FUNCTION_BLOCK FB_HwRefStopButton
VAR_INPUT
END_VAR
VAR_OUTPUT
END_VAR
VAR
	bInput AT %I* : BOOL;
	bFTrig : F_TRIG;
END_VAR
VAR PERSISTENT
	bDisabled : BOOL := TRUE;
END_VAR

bFTrig(CLK:= (bInput OR bDisabled));

PROPERTY P_bDisabled : BOOL
GET
P_bDisabled := bDisabled;
END_GET
SET
bDisabled := P_bDisabled;
fbSettings.M_WritePersData();
END_SET
END_PROPERTY

PROPERTY P_bReleased : BOOL
GET
P_bReleased := bInput OR bDisabled;
END_GET
END_PROPERTY

PROPERTY P_bTriggered : BOOL
GET
P_bTriggered := bFTrig.Q;
END_GET
END_PROPERTY

END_FUNCTION_BLOCK

(* stored: Version 1.1.0.1, ProductVersion 3.1.4022.10
   POU FB_HwRefStopButton: Id {7baece8b-1dc9-4d4b-a35a-8bb7f3010af5}, SpecialFunc None
   Property P_bDisabled: Id {9a391eb1-fa82-4c73-b410-4c29b5333069}
   Get Get: Id {4a5587e0-93b5-4bb2-8de4-dc9ea1a2a49d}
   Set Set: Id {6e392f9c-69a4-46e7-9d7d-d07a24652417}
   Property P_bReleased: Id {d1645a9a-8a8c-4d35-80e4-186646dba8ce}
   Get Get: Id {32973aaa-590a-4665-8edd-e2bd0a458bae}
   Property P_bTriggered: Id {0d76184b-de85-4a43-a058-c25823b210f0}
   Get Get: Id {a2f4313e-0f34-43e8-b91c-4967decc4811} *)
